(* PLC project Programme MGS_2-07_refactorJOY.project, CODESYS CODESYS V3.5 SP19 Patch 1 *)
(* stored: creationDateTime 2026-06-29T23:37:40.9216594, modificationDateTime 2026-06-29T22:49:33.424 *)

FUNCTION_BLOCK FB_MultiStage_Relay
  VAR_INPUT
    Cmd_Pct : REAL;  (* Consigne finale de l'axe (ex: Y_Pct_Ramped, entre -100.0 et 100.0) *)
    Stage1 : REAL;  (* Seuil d'activation Vitesse 1 (ex: 15.0) *)
    Stage2 : REAL;  (* Seuil d'activation Vitesse 2 (ex: 40.0) *)
    Stage3 : REAL;  (* Seuil d'activation Vitesse 3 (ex: 70.0) *)
    Stage4 : REAL;  (* Seuil d'activation Vitesse 4 (ex: 90.0) *)
  END_VAR
  VAR_OUTPUT
    Q1 : BOOL;  (* Sortie physique Relais Vitesse 1 *)
    Q2 : BOOL;  (* Sortie physique Relais Vitesse 2 *)
    Q3 : BOOL;  (* Sortie physique Relais Vitesse 3 *)
    Q4 : BOOL;  (* Sortie physique Relais Vitesse 4 *)
  END_VAR
  VAR
    AbsCmd : REAL;  (* Variable de travail interne (Valeur absolue) *)
  END_VAR

            // 1. On prend la valeur absolue (Valable en marche avant comme arrière)
AbsCmd := ABS(Cmd_Pct);

// 2. Logique cumulative (Cascade)
Q1 := (AbsCmd >= Stage1);
Q2 := (AbsCmd >= Stage2);
Q3 := (AbsCmd >= Stage3);
Q4 := (AbsCmd >= Stage4);
          
END_FUNCTION_BLOCK
